Fanuc KAREL source: kt00602.KL

-- PROVISIONAL review KL for V1013-1; original PC SHA256 5a28b247f25af7a490d2c3765ab7616787c6867580aadbf4125ffb48b2b517e3
-- Incomplete behavior may be omitted. Consult companion uncertainty JSON. Do not deploy.
PROGRAM KT00602
%NOLOCKGROUP
VAR
  I1 : INTEGER
  I2 : INTEGER
  OUT : REAL
BEGIN
  -- UNRESOLVED_PC offsets 5-16; opcodes 2E,23
  -- UNRESOLVED_PC offsets 21-32; opcodes 2E,23
  -- UNRESOLVED_PC offsets 37-48; opcodes 2E,23
  -- UNRESOLVED_PC offsets 53-64; opcodes 2E,23
  -- UNRESOLVED_PC offsets 69-82; opcodes 21,64,23
  -- UNRESOLVED_PC offsets 87-91; opcodes 7F
END KT00602
